Fanuc KAREL source: kt00923.KL

PROGRAM KT00923
%NOLOCKGROUP
VAR
S1 : STRING[80];S2 : STRING[80];OUT : STRING[80]
BEGIN
--
--
S1='A'
S2='B'
S1='A'
S2='B'
OUT=SUB_STR(S1,1,1)
END KT00923
